TYPE csp_transfer_infeed_barcode_connection_status_enum :
(
	INFEED_BARCODE_CONNECTION_STATUS_OPENING_SOCKET								:=  0,
	INFEED_BARCODE_CONNECTION_STATUS_SOCKET_OPENED								:=  10,
	INFEED_BARCODE_CONNECTION_STATUS_ENABLE_REQUEST 							:=  20,
	INFEED_BARCODE_CONNECTION_STATUS_SEND_BRAND_CONFIG 							:=  25,
	INFEED_BARCODE_CONNECTION_STATUS_CLEAR_PREVIOUS_READ 						:=  28,
	INFEED_BARCODE_CONNECTION_STATUS_ENABLED									:=  30,
	INFEED_BARCODE_CONNECTION_STATUS_TEACH_IN_PROCESS							:=  35,
	INFEED_BARCODE_CONNECTION_STATUS_RUN_MODE_WAITING_FOR_TRIGGER				:=  40,
	INFEED_BARCODE_CONNECTION_STATUS_CLEAN_PREVIOUS_READ_DATA					:=  50,
	INFEED_BARCODE_CONNECTION_STATUS_WAIT_FOR_READY								:=  60,
	INFEED_BARCODE_CONNECTION_STATUS_SPARE_1									:=  70,
	INFEED_BARCODE_CONNECTION_STATUS_ERROR										:=  666
) := INFEED_BARCODE_CONNECTION_STATUS_OPENING_SOCKET;
END_TYPE

(* stored: Version 1.1.0.1, ProductVersion 3.1.4024.3
   DUT csp_transfer_infeed_barcode_connection_status_enum: Id {e0276a05-b55c-095d-22e4-083d1ced9580} *)
